FUNCTION_BLOCK F_LEFT (* leftmost L characters of IN *)
  PACKAGE iec61131::charString;
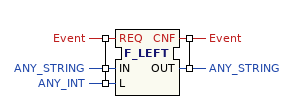
  EVENT_INPUT
    REQ WITH IN, L; (* Service Request *)
  END_EVENT
  EVENT_OUTPUT
    CNF WITH OUT; (* Confirmation of Requested Service *)
  END_EVENT
  VAR_INPUT
    IN : ANY_STRING; (* input string *)
    L : ANY_INT; (* sub-string end position *)
  END_VAR
  VAR_OUTPUT
    OUT : ANY_STRING; (* sub-string from 1 to L *)
  END_VAR
END_FUNCTION_BLOCK
